{attribute addProperty BoxType "IODEVICETYPE_ETHERCATPROT"}
{attribute addProperty Id "TcTerminals210_1EK1100TcTerminals210_1EK1100_99191ECD00SyncUnitsSyncUnits_CAB22D3B19524.375InputsInputs_C75D3FEC1280160OutputsOutputs_47D1E803848106InfoDataInfoData_E9F65A829612"}
{attribute addProperty CRC "3097259386"}
{attribute addProperty SizeInBites "2419"}
{attribute addProperty SizeInBytes "302.375"}
TYPE EtherCAT_Master_KLxxxx_1_B89C6D7A :
STRUCT
	{attribute addProperty Name "TcTerminals210_1EK1100"}
	TcTerminals210_1EK1100 : TcTerminals210_1EK1100_99191ECD;
	{attribute addProperty Name "SyncUnits"}
	SyncUnits : SyncUnits_CAB22D3B;
	{attribute addProperty Name "Inputs"}
	Inputs : Inputs_C75D3FEC;
	{attribute addProperty Name "Outputs"}
	Outputs : Outputs_47D1E803;
	{attribute addProperty Name "InfoData"}
	InfoData : InfoData_E9F65A82;
END_STRUCT
END_TYPE

(* stored: Version 1.2.0.0, ProductVersion 3.1.4024.9
   DUT EtherCAT_Master_KLxxxx_1_B89C6D7A: Id {899dcd3b-1cc5-4b4b-9759-e66c38cf9ea5} *)
